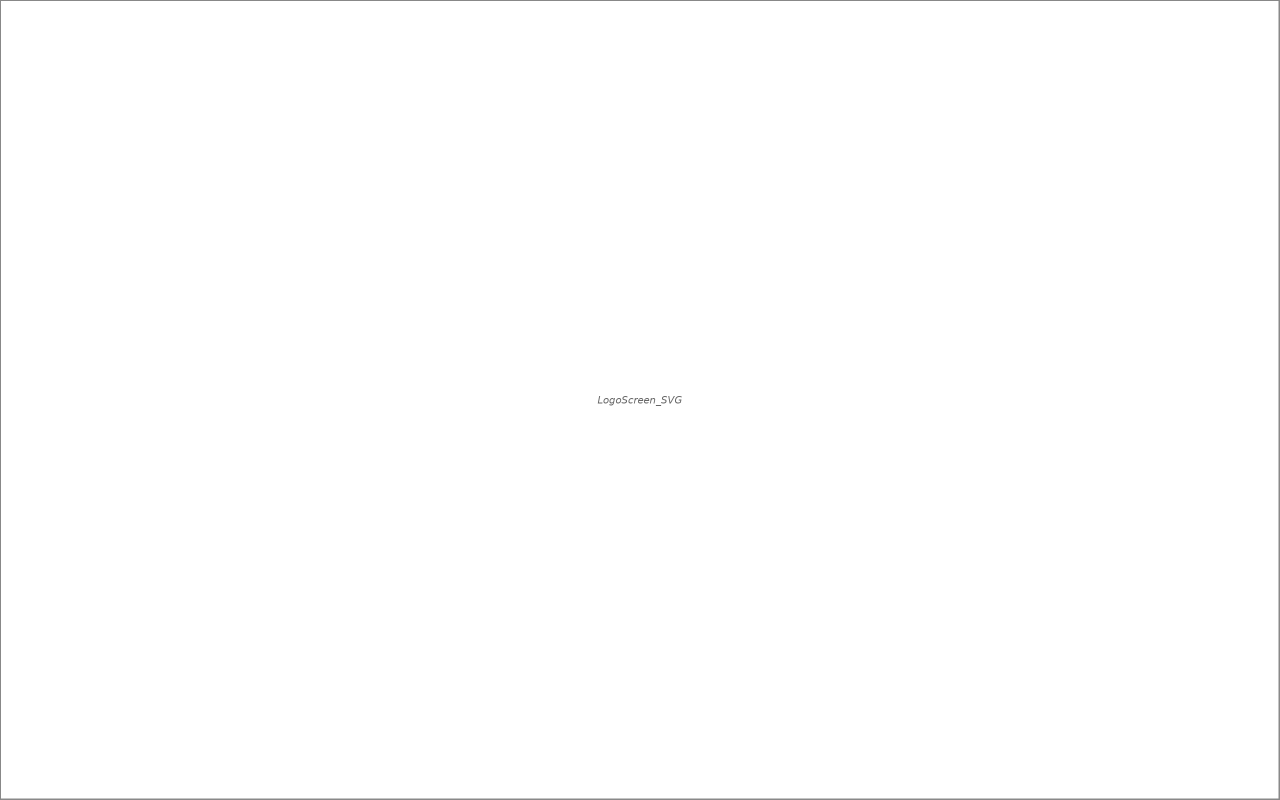
VISUALIZATION Idle  // 1280x800
    Frame (0,0 1280x800), frame switch variable: GVL_HMI.nStartVisu
        shows LogoScreen_SVG()
        shows Settings()
        shows ParameterScreen()
        shows Run()
END_VISUALIZATION

(* stored: Version 1.1.0.1, ProductVersion 3.1.4024.5
   Visu Idle: Id {9c0dfbb2-ead7-41c1-9ffd-e66a861a7940} *)
